FUNCTION_BLOCK INTERNAL FB_Wago750354_BusCoupler
VAR_INPUT
//	b_KbusCycleOverrunFlagDisable			AT %Q* : BOOL;
//	b_InputProcessDataHoldRequest			AT %Q* : BOOL;
//	b_OutputProcessDataHoldRequest			AT %Q* : BOOL;
//	b_OutputDataClearRequest				AT %Q* : BOOL;
	
	b_AckDiagnostics						: BOOL;
	b_ClearDiagnostics						: BOOL;
END_VAR
VAR_OUTPUT
//	b_kBusCycleOverRun						AT %I* : BOOL;
//	b_InputProcessDataHoldAck				AT %I* : BOOL;
//	b_OutputProcessDataHoldAck				AT %I* : BOOL;
//	b_OutputProcessDataClearAck				AT %I* : BOOL;
//	b_NewMessageAvailable					AT %I* : BOOL;
	get											  : ST_Wago750354_get;
END_VAR
VAR	
	ui_DiagnosticsStatusWord			AT %I* : UINT;
	ui_State							AT %I* : UINT;
	DiagnosticsControlWord				AT %Q* : UINT;
END_VAR

get.b_SlaveReady := ui_State = 8;

END_FUNCTION_BLOCK

(* stored: Version 1.1.0.1, ProductVersion 3.1.4024.12
   POU FB_Wago750354_BusCoupler: Id {a3eaf8fd-93ad-4046-9f1d-fb7a9e737f06}, SpecialFunc None *)
